(* IEC 61131-3 sources: Tata_InnoVent/vplc/tasks, 6 files *)

(* ---- furnace.st ---- *)
(* furnace: furnace-1's power controller interface (LOG-100), machine k = 0 on rail psu-b.
   RUN is heat enable. SPEED_PCT is the power limit in %, from DERATE_PCT (%MW10).
   HEAT_ENABLE (%MW21) = 0 turns the heat off. The coil cooling water trip stays in the separate
   OpenPLC interlock. NFPA 86 wants the excess-temperature limit on its own sensor and its own
   device, so it is never part of this controller. *)
PROGRAM furnace
  VAR
    furnace_ready AT %IX0.0 : BOOL;
    furnace_run   AT %QX0.0 : BOOL;
    furnace_power AT %QW0   : INT;
    cell_enable   AT %MW8   : INT := 1;
    power_limit   AT %MW10  : INT := 100;
    heat_enable   AT %MW21  : INT := 1;
  END_VAR
  VAR
    enabled : BOOL;
  END_VAR

  enabled := INT_TO_BOOL(cell_enable) AND INT_TO_BOOL(heat_enable);
  IF furnace_ready AND enabled THEN
    furnace_run := TRUE;
    furnace_power := LIMIT(0, power_limit, 100);
  ELSE
    furnace_run := FALSE;
    furnace_power := 0;
  END_IF;
END_PROGRAM

CONFIGURATION furnace_config
  RESOURCE res0 ON PLC
    TASK main_task(INTERVAL := T#100ms, PRIORITY := 0);
    PROGRAM furn WITH main_task : furnace;
  END_RESOURCE
END_CONFIGURATION

(* ---- machining.st ---- *)
(* machining: the line PLC's interface to cnc-1 (LOG-100), machine k = 0 on rail psu-a.
   A CNC keeps its own controller for the part program, the spindle, and the doors. The line
   PLC sends it the handshake a cell uses: feed enable (off is a feed hold) and the feed override.
   RUN is feed enable. SPEED_PCT is the feed override in %, from DERATE_PCT (%MW10). A CNC allows
   150 % or more. The line keeps it at 0..100 %. FEED_HOLD (%MW21) = 1 holds the feed. *)
PROGRAM machining
  VAR
    cnc_ready    AT %IX0.0 : BOOL;
    cnc_run      AT %QX0.0 : BOOL;
    cnc_speed    AT %QW0   : INT;
    cell_enable  AT %MW8   : INT := 1;
    cnc_override AT %MW10  : INT := 100;
    feed_hold    AT %MW21  : INT := 0;
  END_VAR
  VAR
    enabled : BOOL;
  END_VAR

  enabled := INT_TO_BOOL(cell_enable) AND NOT INT_TO_BOOL(feed_hold);
  IF cnc_ready AND enabled THEN
    cnc_run := TRUE;
    cnc_speed := LIMIT(0, cnc_override, 100);
  ELSE
    cnc_run := FALSE;
    cnc_speed := 0;
  END_IF;
END_PROGRAM

CONFIGURATION machining_config
  RESOURCE res0 ON PLC
    TASK main_task(INTERVAL := T#100ms, PRIORITY := 0);
    PROGRAM mach WITH main_task : machining;
  END_RESOURCE
END_CONFIGURATION

(* ---- packaging-cell-rush.st ---- *)
(* packaging-cell-rush: the packaging cell at rush cadence. Same wiring as packaging-cell.
   The wrapper cycles 10 s on and 5 s off, so the electrical load changes twice as often.
   The conveyor runs while the cell is enabled and the conveyor is READY. The labeler follows the
   wrapper. A CTU counts one pack each time a wrap cycle ends. *)
PROGRAM packaging_cell_rush
  VAR
    conveyor_ready  AT %IX0.0 : BOOL;
    wrapper_ready   AT %IX0.1 : BOOL;
    labeler_ready   AT %IX0.2 : BOOL;
    conveyor_run    AT %QX0.0 : BOOL;
    wrapper_run     AT %QX0.1 : BOOL;
    labeler_run     AT %QX0.2 : BOOL;
    conveyor_speed  AT %QW0   : INT;
    wrapper_speed   AT %QW1   : INT;
    labeler_speed   AT %QW2   : INT;
    cell_enable     AT %MW8   : INT := 1;
    conveyor_derate AT %MW10  : INT := 100;
    wrapper_derate  AT %MW11  : INT := 100;
    labeler_derate  AT %MW12  : INT := 100;
    pack_count      AT %MW20  : INT;
    step_word       AT %MW21  : INT;   (* 1 = wrapping, 2 = wrapper pause *)
  END_VAR
  VAR CONSTANT
    STEP_WRAP  : INT := 1;
    STEP_PAUSE : INT := 2;
    WRAP_ON    : TIME := T#10s;
    WRAP_OFF   : TIME := T#5s;
  END_VAR
  VAR
    step       : INT := 1;
    line_ok    : BOOL;
    wrap_time  : TON;
    pause_time : TON;
    packs      : CTU;
  END_VAR

  line_ok := INT_TO_BOOL(cell_enable) AND conveyor_ready;

  CASE step OF
    STEP_WRAP:
      wrap_time(IN := line_ok AND wrapper_ready, PT := WRAP_ON);
      IF wrap_time.Q THEN
        wrap_time(IN := FALSE);
        step := STEP_PAUSE;
      END_IF;
    STEP_PAUSE:
      pause_time(IN := line_ok, PT := WRAP_OFF);
      IF pause_time.Q THEN
        pause_time(IN := FALSE);
        step := STEP_WRAP;
      END_IF;
  ELSE
    step := STEP_WRAP;
  END_CASE;

  packs(CU := step = STEP_PAUSE, R := FALSE, PV := 32767);
  pack_count := packs.CV;
  step_word := step;

  conveyor_run := line_ok;
  wrapper_run := line_ok AND wrapper_ready AND step = STEP_WRAP;
  labeler_run := wrapper_run AND labeler_ready;

  IF conveyor_run THEN conveyor_speed := LIMIT(0, conveyor_derate, 100); ELSE conveyor_speed := 0; END_IF;
  IF wrapper_run THEN wrapper_speed := LIMIT(0, wrapper_derate, 100); ELSE wrapper_speed := 0; END_IF;
  IF labeler_run THEN labeler_speed := LIMIT(0, labeler_derate, 100); ELSE labeler_speed := 0; END_IF;
END_PROGRAM

CONFIGURATION packaging_rush_config
  RESOURCE res0 ON PLC
    TASK main_task(INTERVAL := T#100ms, PRIORITY := 0);
    PROGRAM packaging WITH main_task : packaging_cell_rush;
  END_RESOURCE
END_CONFIGURATION

(* ---- packaging-cell.st ---- *)
(* packaging-cell: conveyor, wrapper, labeler (machine index k = 0, 1, 2 per FLEET.md 3.1).
   The conveyor runs while the cell is enabled and the conveyor is READY.
   The wrapper cycles WRAP_ON on and WRAP_OFF off. The labeler follows the wrapper.
   A CTU counts one pack each time a wrap cycle ends. Speeds follow the DERATE_PCT setpoints. *)
PROGRAM packaging_cell
  VAR
    conveyor_ready  AT %IX0.0 : BOOL;
    wrapper_ready   AT %IX0.1 : BOOL;
    labeler_ready   AT %IX0.2 : BOOL;
    conveyor_run    AT %QX0.0 : BOOL;
    wrapper_run     AT %QX0.1 : BOOL;
    labeler_run     AT %QX0.2 : BOOL;
    conveyor_speed  AT %QW0   : INT;
    wrapper_speed   AT %QW1   : INT;
    labeler_speed   AT %QW2   : INT;
    cell_enable     AT %MW8   : INT := 1;
    conveyor_derate AT %MW10  : INT := 100;
    wrapper_derate  AT %MW11  : INT := 100;
    labeler_derate  AT %MW12  : INT := 100;
    pack_count      AT %MW20  : INT;
    step_word       AT %MW21  : INT;   (* 1 = wrapping, 2 = wrapper pause *)
  END_VAR
  VAR CONSTANT
    STEP_WRAP  : INT := 1;
    STEP_PAUSE : INT := 2;
    WRAP_ON    : TIME := T#20s;
    WRAP_OFF   : TIME := T#10s;
  END_VAR
  VAR
    step       : INT := 1;
    line_ok    : BOOL;
    wrap_time  : TON;
    pause_time : TON;
    packs      : CTU;
  END_VAR

  line_ok := INT_TO_BOOL(cell_enable) AND conveyor_ready;

  CASE step OF
    STEP_WRAP:
      wrap_time(IN := line_ok AND wrapper_ready, PT := WRAP_ON);
      IF wrap_time.Q THEN
        wrap_time(IN := FALSE);
        step := STEP_PAUSE;
      END_IF;
    STEP_PAUSE:
      pause_time(IN := line_ok, PT := WRAP_OFF);
      IF pause_time.Q THEN
        pause_time(IN := FALSE);
        step := STEP_WRAP;
      END_IF;
  ELSE
    step := STEP_WRAP;
  END_CASE;

  packs(CU := step = STEP_PAUSE, R := FALSE, PV := 32767);
  pack_count := packs.CV;
  step_word := step;

  conveyor_run := line_ok;
  wrapper_run := line_ok AND wrapper_ready AND step = STEP_WRAP;
  labeler_run := wrapper_run AND labeler_ready;

  IF conveyor_run THEN conveyor_speed := LIMIT(0, conveyor_derate, 100); ELSE conveyor_speed := 0; END_IF;
  IF wrapper_run THEN wrapper_speed := LIMIT(0, wrapper_derate, 100); ELSE wrapper_speed := 0; END_IF;
  IF labeler_run THEN labeler_speed := LIMIT(0, labeler_derate, 100); ELSE labeler_speed := 0; END_IF;
END_PROGRAM

CONFIGURATION packaging_config
  RESOURCE res0 ON PLC
    TASK main_task(INTERVAL := T#100ms, PRIORITY := 0);
    PROGRAM packaging WITH main_task : packaging_cell;
  END_RESOURCE
END_CONFIGURATION

(* ---- stamping-line.st ---- *)
(* stamping-line: the base stamping cell (press-1, press-2 on rail psu-a).
   Both presses run all the time. Each press runs at SPEED_PCT = LIMIT(0, DERATE_PCT, 100)
   while it is READY (not tripped) and CELL_ENABLE is 1. Otherwise RUN is off and SPEED_PCT is 0.
   Wiring follows FLEET.md 3.1 with machine index k: press-1 is k = 0, press-2 is k = 1. *)
PROGRAM stamping_line
  VAR
    press1_ready  AT %IX0.0 : BOOL;
    press2_ready  AT %IX0.1 : BOOL;
    press1_amps   AT %IW0   : INT;   (* A x10 *)
    press1_temp   AT %IW1   : INT;   (* degC x10 *)
    press1_volts  AT %IW2   : INT;   (* V x10 *)
    press1_thru   AT %IW3   : INT;   (* pct x10 *)
    press2_amps   AT %IW4   : INT;
    press2_temp   AT %IW5   : INT;
    press2_volts  AT %IW6   : INT;
    press2_thru   AT %IW7   : INT;
    press1_run    AT %QX0.0 : BOOL;
    press2_run    AT %QX0.1 : BOOL;
    press1_speed  AT %QW0   : INT;
    press2_speed  AT %QW1   : INT;
    cell_enable   AT %MW8   : INT := 1;
    press1_derate AT %MW10  : INT := 100;
    press2_derate AT %MW11  : INT := 100;
    running_count AT %MW20  : INT;   (* presses commanded to run this scan *)
  END_VAR
  VAR
    enabled : BOOL;
  END_VAR

  enabled := INT_TO_BOOL(cell_enable);

  IF press1_ready AND enabled THEN
    press1_run := TRUE;
    press1_speed := LIMIT(0, press1_derate, 100);
  ELSE
    press1_run := FALSE;
    press1_speed := 0;
  END_IF;

  IF press2_ready AND enabled THEN
    press2_run := TRUE;
    press2_speed := LIMIT(0, press2_derate, 100);
  ELSE
    press2_run := FALSE;
    press2_speed := 0;
  END_IF;

  running_count := BOOL_TO_INT(press1_run) + BOOL_TO_INT(press2_run);
END_PROGRAM

CONFIGURATION stamping_config
  RESOURCE res0 ON PLC
    TASK main_task(INTERVAL := T#100ms, PRIORITY := 0);
    PROGRAM stamping WITH main_task : stamping_line;
  END_RESOURCE
END_CONFIGURATION

(* ---- utilities.st ---- *)
(* utilities: the plant utilities PLC (LOG-100). compressor-1 is machine k = 0 and chiller-1 is
   k = 1, both on rail psu-b (FLEET.md 3.1). Instruments from the field port: %IW32 the compressor
   pressure transducer (bar x100), %IW33 the loop supply temperature (C x10), %IW34 the loop flow
   (L/min x10), %IW35 the chiller load (% x10).
   compressor-1: a load/unload band on the transducer reading, as a compressor controller runs it
   (Atlas Copco recommends at least 0.6 bar between load and unload). It loads at or below LOAD_P
   and unloads at or above UNLOAD_P. SPEED_PCT is the load: 100 loaded, 25 unloaded. Its
   DERATE_PCT (%MW10) is the run command: 0 stops it, 1..100 runs it. After a stop it waits
   MIN_STOP before it may run again (the controller's minimum stop time).
   chiller-1: runs while the cell is enabled, it is READY (its overload relay is closed), and its
   DERATE_PCT (%MW11) is above 0. SPEED_PCT is that value: the demand limit in % of capacity.
   The chiller's own unit controller keeps its anti-recycle timer. *)
PROGRAM utilities
  VAR
    comp_ready     AT %IX0.0 : BOOL;
    chiller_ready  AT %IX0.1 : BOOL;
    air_p          AT %IW32  : INT;   (* bar x100, the transducer reading *)
    supply_t       AT %IW33  : INT;   (* C x10 *)
    loop_flow      AT %IW34  : INT;   (* L/min x10 *)
    chiller_load   AT %IW35  : INT;   (* % x10 *)
    comp_run       AT %QX0.0 : BOOL;
    chiller_run    AT %QX0.1 : BOOL;
    comp_speed     AT %QW0   : INT;
    chiller_speed  AT %QW1   : INT;
    cell_enable    AT %MW8   : INT := 1;
    comp_cmd       AT %MW10  : INT := 100;
    chiller_limit  AT %MW11  : INT := 100;
    load_p         AT %MW21  : INT := 690;   (* bar x100 *)
    unload_p       AT %MW22  : INT := 750;   (* bar x100 *)
    loaded_word    AT %MW23  : INT;          (* 1 while the compressor is loaded *)
  END_VAR
  VAR CONSTANT
    MIN_STOP : TIME := T#120s;
    UNLOADED : INT := 25;
  END_VAR
  VAR
    enabled     : BOOL;
    loaded      : BOOL;
    comp_on     : BOOL := TRUE;    (* a PLC restart does not stop a running compressor *)
    stopped_for : TON;
  END_VAR

  enabled := INT_TO_BOOL(cell_enable);

  (* the run command, with the minimum stop time before a restart *)
  stopped_for(IN := NOT comp_on, PT := MIN_STOP);
  IF enabled AND comp_ready AND comp_cmd > 0 THEN
    IF NOT comp_on AND stopped_for.Q THEN
      comp_on := TRUE;
    END_IF;
  ELSE
    comp_on := FALSE;
  END_IF;

  (* the load/unload band on the transducer reading *)
  IF comp_on THEN
    IF air_p <= load_p THEN
      loaded := TRUE;
    END_IF;
    IF air_p >= unload_p THEN
      loaded := FALSE;
    END_IF;
  ELSE
    loaded := FALSE;
  END_IF;

  comp_run := comp_on;
  IF comp_on THEN
    IF loaded THEN
      comp_speed := 100;
    ELSE
      comp_speed := UNLOADED;
    END_IF;
  ELSE
    comp_speed := 0;
  END_IF;
  loaded_word := BOOL_TO_INT(loaded);

  chiller_run := enabled AND chiller_ready AND chiller_limit > 0;
  IF chiller_run THEN
    chiller_speed := LIMIT(0, chiller_limit, 100);
  ELSE
    chiller_speed := 0;
  END_IF;
END_PROGRAM

CONFIGURATION utilities_config
  RESOURCE res0 ON PLC
    TASK main_task(INTERVAL := T#100ms, PRIORITY := 0);
    PROGRAM util WITH main_task : utilities;
  END_RESOURCE
END_CONFIGURATION
